PROGRAM MAIN
VAR
	// Safety / Estop override
	bEnabled: BOOL;							// manually turn off / disable output 

	// Temp control FB vars
	fbTempContrl: FB_CTRL_TempController;	
	nControllerMode: E_CTRL_MODE;			// := eCTRL_MODE_TUNE; (* start with tuning *)
	bHeaterOn: BOOL;						// PWM digital output
	rTempF: REAL;							// Actual temperature feedback
	
	fSetPoint: REAL :=100.0;				// if using tuning, setpoint must be > .8 of (initial + tuning step)
	bHeat: BOOL;							// output of controller 

	// simulation model vars
	rTempBuf: ARRAY[1..iMaxDelay] OF REAL; 	// array for delay
	iDelay: UINT:=500;						// thermal temp delay --> 500 is 5 sec
	rHeatGain: REAL := 0.05;				// how big is heater
	rCoolOffGain: REAL := 0.0001;			// ambient cooling effect
	bResetModel: BOOL;						// reset model to zero
	
	// tuning PID gains
	sParaControlExternal	: ST_CTRL_ParaController := (
		// for use when NOT starting with tuning -- values need
		// to be calc'd or determined once with autotuning Controller parameter set - heating 
		KpHeat			:= 32.36,
		TnHeat			:= T#51S502MS,
		TvHeat			:= T#10S815MS,
		TdHeat			:= T#2S704MS,

		// Controller parameter set - cooling - not used in this example
		KpCool			:= 0,
		TnCool			:= T#0S,
		TvCool			:= T#0S,
		TdCool			:= T#0S
		);


	// controller parameter struct (populated)
	stCntrlParam	: ST_CTRL_TempCtrlParameter := (		
		
		(* general parameters 													 *)
		iMode					:= 1,											(* 1=heating, 2=cooling, 3=heating&cooling *)
		iReactionOnFailure		:= eCTRL_ReactionOnFailure_StopController,		(* 0=controller off, 1=manual op, 2=yMin, 3=yMax *)
	
		bSelCtrlParameterSet	:= FALSE,										(* FALSE = internal set, TRUE = external set *)
	
		dwAlarmSupp				:= 16#0000EFFF,									(* alarm suppression *)
		tCtrlCycleTime			:= T#500MS,										(* controller cycle time *)
		tTaskCycleTime			:= T#10MS,										(* plc task cycle time *)
		
		(* tuning parameters 													 *)
		iTuningMode				:= 1,											(* only heating, only cooling, first heating then cooling or vice versa *)
	
		tTuneStabilisation		:= T#20S,										(* wait for a stable system *)
	
		fEndTunePercentHeating	:= 80.0,										(* switch to closed loop control when X > 0.8*W *)
		fYTuneHeating			:= 100.0,										(* step change while tuning operation *)
		fYStableHeating			:= 0.0,											(* tuning operation *)
	
		fEndTunePercentCooling	:= 20.0,										(* switch to closed loop control when X < 0.2*W *)
		fYTuneCooling			:= 0.0,											(* step change while tuning operation *)
		fYStableCooling			:= 0.0,											(* tuning operation *)
		fScalingFactor			:= 1.0,											(* Scaling factor for KP heating/cooling *)
		
		(* setpoint parameters 													 *)
		fWMin					:= 0.0,											(* lower limit *)
		fWMax					:= 300.0,										(* upper limit *)
	
		(* start up *)
		bEnableSoftStart		:= FALSE,										(* FALSE = no soft start, TRUE = soft start *)
		bEnableRamping			:= FALSE,										(* FALSE = no ramping, TRUE = ramping *)
	
		fWStartUp				:= 0.0,											(* soft start plateau setpoint *)
		tStartUp				:= T#0MS,										(* soft start waiting time*)
		bStartUpRamping			:= FALSE,										(* enable ramping while start up phase *)
		fWStartUpVeloPos		:= 1.0,											(* max gradient for increasing setpoint in start up phase*)
		fWStartUpVeloNeg		:= 1.0,											(* max gradient for decreasing setpoint in start up phase *)
	
		fWVeloPos				:= 1.0,											(* max gradient for increasing setpoint *)
		fWVeloNeg				:= 1.0,											(* max gradient for decreasing setpoint *)	
	
		(* actual value parameters     											 *)
		bFilter 				:= FALSE,
		tFilter					:= T#0S,
		
		(* deadband parameters     												 *)
		bDeadband				:= FALSE,
		fEDeadband				:= 0.0,											(* deadband *)
		
		(* control value parameters     										 *)
		fYMin					:= 0.0,											(* lower limit *)
		fYMax					:= 100.0,										(* upper limit *)
		fYManual				:= 0.0,									 		(* manual operation*)
		fYOnFailure				:= 0.0,											(* control value on failure *)
	
		tPWMCycleTime			:= t#1s,										(* PWM: period *)
		tPWMMinOffTime			:= t#0s,										(* PWM: min off time *)
		tPWMMinOnTime			:= t#0s,										(* PWM: min on time *)
		tPWMWaitingTime			:= t#0s,										(* PWM: min waiting time *) (* not yet implemented !!!!*)
	
		fYThresholdOff			:= 0.0,											(* 3-Point: Off threshold *)
		fYThresholdOn			:= 0.0,											(* 3-Point: On threshold *)
	
		nCyclesForSwitchOver	:= 100,
	
		(* controller settings			     									 *)
		bEnablePreController 	:= FALSE,										(* enable precontroller *)
		bEnableZones 			:= FALSE,										(* enable zone around setpoint with open loop control *)
		bEnableCVFilter 		:= FALSE,										(* enable filter for CV (type see iFilterType) *)
		iFilterType 			:= eCTRL_FilterType_FIRSTORDER,			 		(* filtertype of CV filter *)
		iControllerType 		:= eCTRL_ControllerType_PID,					(* used controller normally PID *)
		
		
		(* min max temperatures	     											 *)
		TempLow					:= -5.0,
		TempLowLow				:= -10.0,
		TempHigh				:= 5.0,
		TempHighHigh			:= 10.0,
		TempAbsoluteHigh		:= 300.0,
		TempAbsoluteLow			:= 0.0,	
		
		(* internal tuning parameters *)
		fTuneKp					:= 1.2,
		fTuneTn					:= 2.0,
		fTuneTv					:= 0.42,
		fTuneTd					:= 0.25
		);
		
	bLoadTuneParamSet			:BOOL;
	SelectedParamSetToLoad		:E_TunePreSets;	
END_VAR
VAR CONSTANT
	TuneParamPreSets: ARRAY [E_TunePreSets.Fast..E_TunePreSets.Asymptotic] OF ST_TuneParams := 
	[	(fKp := 1.2, fTn := 2.0, fTv := 0.42, fTd := 0.25), 
		(fKp := 1.0, fTn := 2.5, fTv := 0.42, fTd := 0.25), 
		(fKp := 0.5, fTn := 3.0, fTv := 1.0, fTd := 0.25)
	];	
	iMaxDelay		:UINT := 6000;	// 6000 is 60 seconds
END_VAR


TempControl();

(* manually disable heater output if needed *)
IF bEnabled AND bHeat THEN
	bHeaterOn := TRUE;
ELSE
	bHeaterOn := FALSE;
END_IF

IF bLoadTuneParamSet THEN
	bLoadTuneParamSet	:=FALSE;
	stCntrlParam.fTuneKp:=TuneParamPreSets[SelectedParamSetToLoad].fKp;
	stCntrlParam.fTuneTd:=TuneParamPreSets[SelectedParamSetToLoad].fTd;
	stCntrlParam.fTuneTn:=TuneParamPreSets[SelectedParamSetToLoad].fTn;
	stCntrlParam.fTuneTv:=TuneParamPreSets[SelectedParamSetToLoad].fTv;
	
END_IF

// simulated process with thermal time delay
rTempBuf[1] := rTempBuf[1] + BOOL_TO_REAL(bHeaterOn)* rHeatGain - (rTempBuf[1]*rCoolOffGain);
rTempF := rTempBuf[iDelay];
MEMCPY(destAddr:= ADR(rTempBuf[2]), srcAddr:= ADR(rTempBuf[1]), n:= (iMaxDelay-1)*SIZEOF(rTempBuf[1]));

IF bResetModel THEN
	bResetModel:=FALSE;
	MEMSET(destAddr:= ADR(rTempBuf[1]), fillByte:= 16#00, n:= (iMaxDelay)*SIZEOF(rTempBuf[1]));
END_IF

ACTION TempControl:
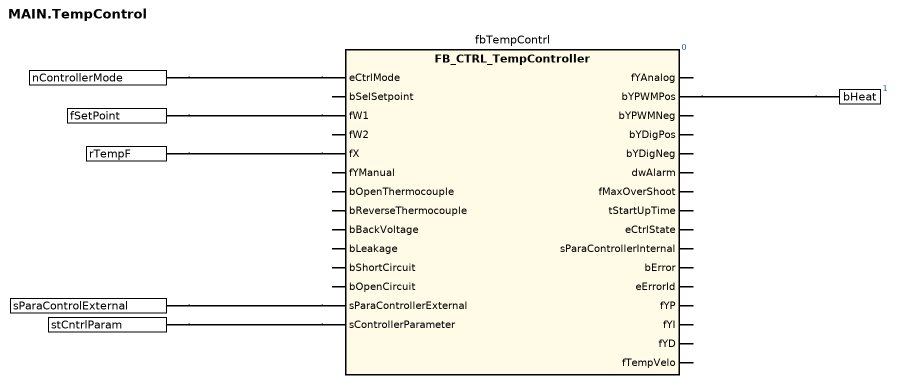
fbTempContrl(
    eCtrlMode := nControllerMode,
    fW1 := fSetPoint,
    fX := rTempF,
    sParaControllerExternal := sParaControlExternal,
    sControllerParameter := stCntrlParam); // FB_CTRL_TempController
bHeat := fbTempContrl.bYPWMPos;
END_ACTION

END_PROGRAM

(* stored: Version 1.1.0.1, ProductVersion 3.1.4024.11
   POU MAIN: Id {b589477e-ee93-40e8-aa5d-96f84a6164c4}, SpecialFunc None
   Action TempControl: Id {bc0f30f8-ea59-4f14-a5ab-fe0e0085fba9} *)
